// Queue Decorator for function blocks that impliment I_List interface
{attribute 'enable_dynamic_creation'}
FUNCTION_BLOCK FB_Queue EXTENDS FB_Collection  IMPLEMENTS I_Queue
VAR_INPUT
	ipList : I_List; // List to perform operations on.
END_VAR

(* Number of items in queue*)
PROPERTY _Count : T_Capacity
GET
IF THIS^.NullReferenceException() THEN _Count := -1;RETURN; END_IF
_Count := THIS^.ipList._Count;
END_GET
END_PROPERTY

PROPERTY _Error_Status : ST_ERROR
GET
IF THIS^.NullReferenceException() THEN _Error_Status := THIS^.stError; RETURN; END_IF
THIS^.stError := THIS^.ipList._Error_Status;
_Error_Status := F_Error(THIS^.stError.bSTATUS, THIS^.stError.nCODE, THIS^.stError.sSOURCE);
END_GET
END_PROPERTY

(* Checks of queue is empty.*)
PROPERTY _Is_Empty : BOOL
GET
IF THIS^.NullReferenceException() THEN _Is_Empty := TRUE; RETURN; END_IF
_Is_Empty := THIS^.ipList._Is_Empty;
END_GET
END_PROPERTY

METHOD PROTECTED CatchError : BOOL
VAR_INPUT
END_VAR
IF THIS^.NullReferenceException() THEN RETURN; END_IF
THIS^.stError := ipList._Error_Status;
CatchError := stError.bSTATUS;
END_METHOD

(* Empties/Clears/Deletes every item on the queue*)
METHOD Clear
IF THIS^.NullReferenceException() THEN RETURN; END_IF
THIS^.ipList.Clear();
END_METHOD

(* Gets and remove item at the front of the queue *)
METHOD Dequeue : I_Queue
VAR_INPUT
	Item : ANY; (* Variable to store returned item value *)
END_VAR
VAR_OUTPUT
	bSuccess : BOOL;
END_VAR
VAR 
	bA, bB 	 : BOOL;
END_VAR
Dequeue := THIS^;
IF THIS^.NullReferenceException() THEN RETURN; END_IF
THIS^.ipList.Get_First(Item, bSuccess => bA);
THIS^.ipList.Remove(bSuccess => bB);
bSuccess := bA AND bB;
END_METHOD

(* Removes item at the front of the queue without returning anything *)
METHOD Dequeue_Void : I_Queue
VAR_OUTPUT
	bSuccess : BOOL;
END_VAR
Dequeue_Void := THIS^;
IF THIS^.NullReferenceException() THEN RETURN; END_IF
THIS^.ipList.Remove(bSuccess => bSuccess);
THIS^.CatchError();
END_METHOD

(* Adds item at the back of the queue *)
METHOD Enqueue : I_Queue
VAR_INPUT
	Item : ANY; (* Variable containg data to store on the queue *)
END_VAR
VAR_OUTPUT
	bSuccess : BOOL;
END_VAR
Enqueue := THIS^;
IF THIS^.NullReferenceException() THEN RETURN; END_IF
THIS^.ipList.Add_Back(Item, bSuccess => bSuccess);
THIS^.CatchError();
END_METHOD

(* Adds item at the front of the queue *)
METHOD Enqueue_At_Front : I_Queue
VAR_INPUT
	Item : ANY; (* Variable containg data to store on the queue *)
END_VAR
VAR_OUTPUT
	bSuccess : BOOL;
END_VAR
Enqueue_At_Front := THIS^;
IF THIS^.NullReferenceException() THEN RETURN; END_IF
THIS^.ipList.Add_Front(Item, bSuccess => bSuccess);
THIS^.CatchError();
END_METHOD

METHOD PROTECTED NullReferenceException : BOOL
NullReferenceException := THIS^.ipList = 0;
IF NOT NullReferenceException THEN RETURN; END_IF
THIS^.RaiseException(2000+GVL_CmpErrors.ERR_INVALID_REFERENCE, 'Null or Invalid Reference');
END_METHOD

(* Get item from the queue without removing it. *)
METHOD Peek : I_Queue
VAR_INPUT
	Item 	: ANY; (* Variable to store returned item value *)
	nIndex 	: DINT; (* Location of item*)
END_VAR
VAR_OUTPUT
	bSuccess : BOOL;
END_VAR
Peek := THIS^;
IF THIS^.NullReferenceException() THEN RETURN; END_IF
THIS^.ipList.Get(Item, nIndex, bSuccess => bSuccess);
THIS^.CatchError();
END_METHOD

METHOD Reverse : I_Queue
VAR_OUTPUT
	bSuccess : BOOL;
END_VAR
Reverse := THIS^;
IF THIS^.NullReferenceException() THEN RETURN; END_IF
THIS^.ipList.Reverse(bSuccess => bSuccess);
THIS^.CatchError();
END_METHOD

END_FUNCTION_BLOCK

(* stored: Version 1.1.0.1, ProductVersion 3.1.4024.4
   POU FB_Queue: Id {c0a25d3b-3294-43fd-9bd2-3bf3486c2d23}, SpecialFunc None
   Folder Exceptions: Id {32400bd4-b7e2-4496-a434-64275e7e67c6}
   Property _Count: Id {4980f9f4-e529-4835-9d02-e0820fac350a}
   Get Get: Id {699f6c1f-1997-44e0-9196-f27626bb4a8b}
   Property _Error_Status: Id {72a39777-456e-4c2e-85d6-936041c24d4c}
   Get Get: Id {66fdd621-1599-41ea-8e13-ba87dc445cb1}
   Property _Is_Empty: Id {b2cc4ea1-9af3-4348-b1a8-14581439c42b}
   Get Get: Id {d0d3dd0b-a078-4014-b6a2-e264180a9714}
   Method CatchError: Id {ff942c32-b1f2-46ab-998e-004a022407f0}
   Method Clear: Id {76443963-9b9c-4996-b3e7-fc775a7561d8}
   Method Dequeue: Id {e93db59e-1376-4260-b5d7-9c96340c297e}
   Method Dequeue_Void: Id {fb75845f-f99c-4e28-94cd-b00a8977d52c}
   Method Enqueue: Id {407277f4-3eec-4c29-a153-3392e4cf9679}
   Method Enqueue_At_Front: Id {b3f4e9ed-60eb-4205-a930-b6e55d94d98e}
   Method NullReferenceException: Id {2f7bb67e-e1e1-4b51-b486-f5636567eb0e}
   Method Peek: Id {bd5b0349-051a-47b0-b681-deca70a87271}
   Method Reverse: Id {379b4de2-5f3c-405e-9591-f9fd46fb229d} *)
